// TIA Portal V19 export
VAR_GLOBAL   // PLC tag table "Comm with 1500"
   Green_from_1500 AT %M0.5 : Bool;
   Red_from_1500 AT %M0.6 : Bool;
   Blue_from_1500 AT %M0.7 : Bool;
   PB_Green_from_1500 AT %M0.0 : Bool;
   PB_Blue_from_1500 AT %M0.1 : Bool;
   OS1 AT %M2.0 : Bool;
   Error1 AT %M2.1 : Bool;
   status1 AT %MW4 : Word;
   history1 AT %MW6 : Word;
   Output_data_from_1500 AT %MB0 : Byte;
   OutputDataFrom1500 AT %MW0 : Word;
   Tag_6 AT %MW52 : Int;
   Input_buffer_to_1500 AT %MD50 : DWord;
END_VAR
